{attribute addProperty BoxType "EK1100-0000-0018"}
{attribute addProperty Id "boxesEK1122boxesEK1122_6347E4412630328.75A_0001_EJ5151_0000_0016EJ5151_0AC1A36D19424.25A_0002_EL1262_0000_0002EL1262_FE5A7D8230638.25A_0003_EL1262_0000_0003EL1262_FE5A7D8230638.25A_0004_EL1262_0050_0002EL1262_FE5A7D8230638.25A_0005_EL1262_0050_0003EL1262_FE5A7D8230638.25A_0006_EL2262_0000_0001EL2262_6FCF2F7B12916.125A_0007_EL2262_0000_0002EL2262_131C31B227334.125A_0008_EL2262_0000_0003EL2262_131C31B227334.125A_0009_EL2262_0000_0004EL2262_E0ACD1AC30638.25A_0010_EL3681_0000_0017EL3681_0CFA3F6116220.25A_0011_EL3681_0000_0018EL3681_BC5DB35D16220.25A_0012_EL3681_0000_0019EL3681_BC5DB35D16220.25A_0013_EL3681_0000_0020EL3681_C596F5D116220.25A_0014_EL5101_0000_0000EL5101_8E82486614618.25A_0015_EL5151_0000_0016EL5151_7DE9C09925832.25A_0016_EL5151_0000_0017EL5151_023DC4F232240.25A_0017_EL5151_0000_0018EL5151_023DC4F232240.25A_0018_EL5151_0000_0019EL5151_023DC4F232240.25A_0019_EL5151_0000_0020EL5151_B6C9029519424.25A_0020_EL5151_0000_0025EL5151_0AC1A36D19424.25A_0021_EL5151_0000_0026EL5151_0AC1A36D19424.25A_0022_EL5151_0080_0016EL5151_09E56EF027434.25A_0023_EL5151_0080_0017EL5151_B6C9029519424.25A_0024_EL5151_0080_0018EL5151_B6C9029519424.25A_0025_EL5151_0080_0019EL5151_B6C9029519424.25A_0026_EL5151_0080_0020EL5151_B6C9029519424.25A_0027_EL5151_0080_0021EL5151_0AC1A36D19424.25A_0028_EL3773_0000_0016EL3773_90A9FC821282160.25A_0029_EM7004_0000_9995EM7004_4021F80C72290.25A_0041_AX8108_0100_0101AX8108_E4DF803355669.5A_0042_AX8108_0100_0102AX8108_5E0E86F855669.5A_0043_AX8108_0100_0103AX8108_5E0E86F855669.5A_0044_AX8108_0100_0104AX8108_5E0E86F855669.5A_0045_AX8108_0110_0102AX8108_5E0E86F855669.5A_0046_AX8108_0110_0103AX8108_5E0E86F855669.5A_0047_AX8108_0110_0104AX8108_5E0E86F855669.5A_0048_AX8108_0200_0103AX8108_5E0E86F855669.5A_0049_AX8108_0200_0104AX8108_5E0E86F855669.5A_0050_AX8108_0210_0103AX8108_5E0E86F855669.5A_0051_AX8108_0210_0104AX8108_5E0E86F855669.5A_0052_AX8118_0100_0101AX8118_E4DF803355669.5A_0053_AX8118_0100_0102AX8118_5E0E86F855669.5A_0054_AX8118_0100_0103AX8118_5E0E86F855669.5A_0055_AX8118_0100_0104AX8118_5E0E86F855669.5A_0056_AX8118_0110_0102AX8118_5E0E86F855669.5A_0057_AX8118_0110_0103AX8118_5E0E86F855669.5A_0058_AX8118_0110_0104AX8118_5E0E86F855669.5A_0059_AX8118_0200_0103AX8118_5E0E86F855669.5A_0060_AX8118_0200_0104AX8118_5E0E86F855669.5A_0061_AX8118_0210_0103AX8118_5E0E86F855669.5A_0062_AX8118_0210_0104AX8118_5E0E86F855669.5A_0063_AX8206_0100_0101AX8206_36A80AF074092.5A_0064_AX8206_0100_0102AX8206_AF8A8AFA74092.5A_0065_AX8206_0100_0103AX8206_AF8A8AFA74092.5A_0066_AX8206_0100_0104AX8206_AF8A8AFA74092.5A_0067_AX8206_0110_0102AX8206_AF8A8AFA74092.5A_0068_AX8206_0110_0103AX8206_AF8A8AFA74092.5A_0069_AX8206_0110_0104AX8206_AF8A8AFA74092.5A_0070_AX8206_0200_0103AX8206_AF8A8AFA74092.5A_0071_AX8206_0200_0104AX8206_AF8A8AFA74092.5A_0072_AX8206_0210_0103AX8206_AF8A8AFA74092.5A_0073_AX8206_0210_0104AX8206_AF8A8AFA74092.5A_0074_EM7004_0000_9995EM7004_4021F80C72290.25A_0075_AX8118_0100_0101AX8118_E4DF803355669.5"}
{attribute addProperty CRC "2974716934"}
{attribute addProperty SizeInBites "32527"}
{attribute addProperty SizeInBytes "4065.875"}
TYPE boxes_B14E9406 EXTENDS EK1100_179A0949 :
STRUCT
	{attribute addProperty Name "boxesEK1122"}
	boxesEK1122 : boxesEK1122_6347E441;
	{attribute addProperty Name "A_0001_EJ5151_0000_0016"}
	A_0001_EJ5151_0000_0016 : EJ5151_0AC1A36D;
	{attribute addProperty Name "A_0002_EL1262_0000_0002"}
	A_0002_EL1262_0000_0002 : EL1262_FE5A7D82;
	{attribute addProperty Name "A_0003_EL1262_0000_0003"}
	A_0003_EL1262_0000_0003 : EL1262_FE5A7D82;
	{attribute addProperty Name "A_0004_EL1262_0050_0002"}
	A_0004_EL1262_0050_0002 : EL1262_FE5A7D82;
	{attribute addProperty Name "A_0005_EL1262_0050_0003"}
	A_0005_EL1262_0050_0003 : EL1262_FE5A7D82;
	{attribute addProperty Name "A_0006_EL2262_0000_0001"}
	A_0006_EL2262_0000_0001 : EL2262_6FCF2F7B;
	{attribute addProperty Name "A_0007_EL2262_0000_0002"}
	A_0007_EL2262_0000_0002 : EL2262_131C31B2;
	{attribute addProperty Name "A_0008_EL2262_0000_0003"}
	A_0008_EL2262_0000_0003 : EL2262_131C31B2;
	{attribute addProperty Name "A_0009_EL2262_0000_0004"}
	A_0009_EL2262_0000_0004 : EL2262_E0ACD1AC;
	{attribute addProperty Name "A_0010_EL3681_0000_0017"}
	A_0010_EL3681_0000_0017 : EL3681_0CFA3F61;
	{attribute addProperty Name "A_0011_EL3681_0000_0018"}
	A_0011_EL3681_0000_0018 : EL3681_BC5DB35D;
	{attribute addProperty Name "A_0012_EL3681_0000_0019"}
	A_0012_EL3681_0000_0019 : EL3681_BC5DB35D;
	{attribute addProperty Name "A_0013_EL3681_0000_0020"}
	A_0013_EL3681_0000_0020 : EL3681_C596F5D1;
	{attribute addProperty Name "A_0014_EL5101_0000_0000"}
	A_0014_EL5101_0000_0000 : EL5101_8E824866;
	{attribute addProperty Name "A_0015_EL5151_0000_0016"}
	A_0015_EL5151_0000_0016 : EL5151_7DE9C099;
	{attribute addProperty Name "A_0016_EL5151_0000_0017"}
	A_0016_EL5151_0000_0017 : EL5151_023DC4F2;
	{attribute addProperty Name "A_0017_EL5151_0000_0018"}
	A_0017_EL5151_0000_0018 : EL5151_023DC4F2;
	{attribute addProperty Name "A_0018_EL5151_0000_0019"}
	A_0018_EL5151_0000_0019 : EL5151_023DC4F2;
	{attribute addProperty Name "A_0019_EL5151_0000_0020"}
	A_0019_EL5151_0000_0020 : EL5151_B6C90295;
	{attribute addProperty Name "A_0020_EL5151_0000_0025"}
	A_0020_EL5151_0000_0025 : EL5151_0AC1A36D;
	{attribute addProperty Name "A_0021_EL5151_0000_0026"}
	A_0021_EL5151_0000_0026 : EL5151_0AC1A36D;
	{attribute addProperty Name "A_0022_EL5151_0080_0016"}
	A_0022_EL5151_0080_0016 : EL5151_09E56EF0;
	{attribute addProperty Name "A_0023_EL5151_0080_0017"}
	A_0023_EL5151_0080_0017 : EL5151_B6C90295;
	{attribute addProperty Name "A_0024_EL5151_0080_0018"}
	A_0024_EL5151_0080_0018 : EL5151_B6C90295;
	{attribute addProperty Name "A_0025_EL5151_0080_0019"}
	A_0025_EL5151_0080_0019 : EL5151_B6C90295;
	{attribute addProperty Name "A_0026_EL5151_0080_0020"}
	A_0026_EL5151_0080_0020 : EL5151_B6C90295;
	{attribute addProperty Name "A_0027_EL5151_0080_0021"}
	A_0027_EL5151_0080_0021 : EL5151_0AC1A36D;
	{attribute addProperty Name "A_0028_EL3773_0000_0016"}
	A_0028_EL3773_0000_0016 : EL3773_90A9FC82;
	{attribute addProperty Name "A_0029_EM7004_0000_9995"}
	A_0029_EM7004_0000_9995 : EM7004_4021F80C;
	{attribute addProperty Name "A_0041_AX8108_0100_0101"}
	A_0041_AX8108_0100_0101 : AX8108_E4DF8033;
	{attribute addProperty Name "A_0042_AX8108_0100_0102"}
	A_0042_AX8108_0100_0102 : AX8108_5E0E86F8;
	{attribute addProperty Name "A_0043_AX8108_0100_0103"}
	A_0043_AX8108_0100_0103 : AX8108_5E0E86F8;
	{attribute addProperty Name "A_0044_AX8108_0100_0104"}
	A_0044_AX8108_0100_0104 : AX8108_5E0E86F8;
	{attribute addProperty Name "A_0045_AX8108_0110_0102"}
	A_0045_AX8108_0110_0102 : AX8108_5E0E86F8;
	{attribute addProperty Name "A_0046_AX8108_0110_0103"}
	A_0046_AX8108_0110_0103 : AX8108_5E0E86F8;
	{attribute addProperty Name "A_0047_AX8108_0110_0104"}
	A_0047_AX8108_0110_0104 : AX8108_5E0E86F8;
	{attribute addProperty Name "A_0048_AX8108_0200_0103"}
	A_0048_AX8108_0200_0103 : AX8108_5E0E86F8;
	{attribute addProperty Name "A_0049_AX8108_0200_0104"}
	A_0049_AX8108_0200_0104 : AX8108_5E0E86F8;
	{attribute addProperty Name "A_0050_AX8108_0210_0103"}
	A_0050_AX8108_0210_0103 : AX8108_5E0E86F8;
	{attribute addProperty Name "A_0051_AX8108_0210_0104"}
	A_0051_AX8108_0210_0104 : AX8108_5E0E86F8;
	{attribute addProperty Name "A_0052_AX8118_0100_0101"}
	A_0052_AX8118_0100_0101 : AX8118_E4DF8033;
	{attribute addProperty Name "A_0053_AX8118_0100_0102"}
	A_0053_AX8118_0100_0102 : AX8118_5E0E86F8;
	{attribute addProperty Name "A_0054_AX8118_0100_0103"}
	A_0054_AX8118_0100_0103 : AX8118_5E0E86F8;
	{attribute addProperty Name "A_0055_AX8118_0100_0104"}
	A_0055_AX8118_0100_0104 : AX8118_5E0E86F8;
	{attribute addProperty Name "A_0056_AX8118_0110_0102"}
	A_0056_AX8118_0110_0102 : AX8118_5E0E86F8;
	{attribute addProperty Name "A_0057_AX8118_0110_0103"}
	A_0057_AX8118_0110_0103 : AX8118_5E0E86F8;
	{attribute addProperty Name "A_0058_AX8118_0110_0104"}
	A_0058_AX8118_0110_0104 : AX8118_5E0E86F8;
	{attribute addProperty Name "A_0059_AX8118_0200_0103"}
	A_0059_AX8118_0200_0103 : AX8118_5E0E86F8;
	{attribute addProperty Name "A_0060_AX8118_0200_0104"}
	A_0060_AX8118_0200_0104 : AX8118_5E0E86F8;
	{attribute addProperty Name "A_0061_AX8118_0210_0103"}
	A_0061_AX8118_0210_0103 : AX8118_5E0E86F8;
	{attribute addProperty Name "A_0062_AX8118_0210_0104"}
	A_0062_AX8118_0210_0104 : AX8118_5E0E86F8;
	{attribute addProperty Name "A_0063_AX8206_0100_0101"}
	A_0063_AX8206_0100_0101 : AX8206_36A80AF0;
	{attribute addProperty Name "A_0064_AX8206_0100_0102"}
	A_0064_AX8206_0100_0102 : AX8206_AF8A8AFA;
	{attribute addProperty Name "A_0065_AX8206_0100_0103"}
	A_0065_AX8206_0100_0103 : AX8206_AF8A8AFA;
	{attribute addProperty Name "A_0066_AX8206_0100_0104"}
	A_0066_AX8206_0100_0104 : AX8206_AF8A8AFA;
	{attribute addProperty Name "A_0067_AX8206_0110_0102"}
	A_0067_AX8206_0110_0102 : AX8206_AF8A8AFA;
	{attribute addProperty Name "A_0068_AX8206_0110_0103"}
	A_0068_AX8206_0110_0103 : AX8206_AF8A8AFA;
	{attribute addProperty Name "A_0069_AX8206_0110_0104"}
	A_0069_AX8206_0110_0104 : AX8206_AF8A8AFA;
	{attribute addProperty Name "A_0070_AX8206_0200_0103"}
	A_0070_AX8206_0200_0103 : AX8206_AF8A8AFA;
	{attribute addProperty Name "A_0071_AX8206_0200_0104"}
	A_0071_AX8206_0200_0104 : AX8206_AF8A8AFA;
	{attribute addProperty Name "A_0072_AX8206_0210_0103"}
	A_0072_AX8206_0210_0103 : AX8206_AF8A8AFA;
	{attribute addProperty Name "A_0073_AX8206_0210_0104"}
	A_0073_AX8206_0210_0104 : AX8206_AF8A8AFA;
	{attribute addProperty Name "A_0074_EM7004_0000_9995"}
	A_0074_EM7004_0000_9995 : EM7004_4021F80C;
	{attribute addProperty Name "A_0075_AX8118_0100_0101"}
	A_0075_AX8118_0100_0101 : AX8118_E4DF8033;
END_STRUCT
END_TYPE

(* stored: Version 1.2.0.0, ProductVersion 3.1.4024.9
   DUT boxes_B14E9406: Id {5f0307c8-6a21-445a-ae63-79e415b1e0c4} *)
